Staubli VAL3: WatchDog.pgx

program WatchDog()
begin
end
